TYPE EL3413_PM_InputsAuxiliaryStatus :
STRUCT
	{attribute 'hide'}
	{attribute addProperty Name "Bit 1(address x.0)"}
	Bit_1 : BIT;
	{attribute 'hide'}
	{attribute addProperty Name "Bit 2(address x.1)"}
	Bit_2 : BIT;
	{attribute addProperty Name "Overcurrent"}
	Overcurrent : BIT;
	{attribute 'hide'}
	{attribute addProperty Name "Bit 4(address x.3)"}
	Bit_4 : BIT;
	{attribute 'hide'}
	{attribute addProperty Name "Bit 5(address x.4)"}
	Bit_5 : BIT;
	{attribute 'hide'}
	{attribute addProperty Name "Bit 6(address x.5)"}
	Bit_6 : BIT;
	{attribute 'hide'}
	{attribute addProperty Name "Bit 7(address x.6)"}
	Bit_7 : BIT;
	{attribute 'hide'}
	{attribute addProperty Name "Bit 8(address x.7)"}
	Bit_8 : BIT;
	{attribute 'hide'}
	{attribute addProperty Name "Bit 9(address x+1.0)"}
	Bit_9 : BIT;
	{attribute 'hide'}
	{attribute addProperty Name "Bit 10(address x+1.1)"}
	Bit_10 : BIT;
	{attribute 'hide'}
	{attribute addProperty Name "Bit 11(address x+1.2)"}
	Bit_11 : BIT;
	{attribute 'hide'}
	{attribute addProperty Name "Bit 12(address x+1.3)"}
	Bit_12 : BIT;
	{attribute 'hide'}
	{attribute addProperty Name "Bit 13(address x+1.4)"}
	Bit_13 : BIT;
	{attribute 'hide'}
	{attribute addProperty Name "Bit 14(address x+1.5)"}
	Bit_14 : BIT;
	{attribute addProperty Name "TxPDO State"}
	TxPDOState : BIT;
	{attribute addProperty Name "TxPDO Toggle"}
	TxPDOToggle : BIT;

END_STRUCT
END_TYPE

(* stored: Version 1.1.0.1, ProductVersion 3.1.4024.9
   DUT EL3413_PM_InputsAuxiliaryStatus: Id {5aa7e1bd-32d2-0df3-0914-57eed10037f8} *)
